(* IEC 61131-3 sources: codesys-build/examples/frame-assembly/src, 1 file *)

(* ---- Main.st ---- *)
PROGRAM Main
VAR
	Station : FB_FramingStation;
END_VAR
PRG_ReadInputs();
PRG_Transport();
Station();
PRG_Publish();
END_PROGRAM
